Fanuc KAREL source: compact_preamble.KL

PROGRAM KA00079
%NOLOCKGROUP
VAR
SRC : XYZWPREXT;DST : XYZWPREXT
BEGIN
SRC.X=1.0
DST=SRC
END KA00079
